{attribute addProperty BoxType "EJ7411-0000-0018"}
{attribute addProperty Id "Following_error_actual_valueAT %I*DINT324"}
{attribute addProperty CRC "4114822454"}
{attribute addProperty SizeInBites "32"}
{attribute addProperty SizeInBytes "4"}
TYPE DRV_Following_error_actual_value_F5433536 :
STRUCT
	{attribute addProperty Name "Following_error_actual_value"}
	Following_error_actual_value AT %I* : DINT;
END_STRUCT
END_TYPE

(* stored: Version 1.2.0.0, ProductVersion 3.1.4024.9
   DUT DRV_Following_error_actual_value_F5433536: Id {00d806bc-3def-4b9d-bc77-f784cf9bb254} *)
